FUNCTION_BLOCK CU00xAutomatParalell_1_Task EXTENDS TcoTaskedSequencer 

VAR
	_customTimer: TON;
END_VAR

Run();

(*~
	<docu>
		<summary>
			Main method of the sequener. Custom code needs to be placed here. The sequencer is executed by call of **Instance.Run()** method.
			This method is abstract, and it must be overridden in derived block.
		</summary>
	</docu>
~*)
METHOD PROTECTED Main : BOOL
// Takes mode (step/continous) from the parent controller
THIS^.ModeController.Mode := ParentSequence.ModeController.Mode;

IF (Step(1000, TRUE, 'PARALELL STEP - EXAMPLE OF TIMERS')) THEN
    //-------------------------------------    
		StepCompleteWhen(CurrentStep.Duration >= T#300mS);	
    //-------------------------------------
END_IF
IF (Step(1100, TRUE, 'PARALELL STEP - EXAMPLE OF TIMERS')) THEN
    //-------------------------------------    
		StepCompleteWhen(inCondition:=Timer_1(TRUE,T#100MS));	
    //-------------------------------------
END_IF
IF (Step(1200, TRUE, 'PARALELL STEP - EXAMPLE OF TIMERS')) THEN
    //-------------------------------------    
		StepCompleteWhen(inCondition:=Timer_1(TRUE,T#200MS));	
    //-------------------------------------
END_IF

IF THIS^.IsFreshState THEN
	_customTimer(IN:=FALSE);
END_IF
IF (Step(1300, TRUE, 'PARALELL STEP - EXAMPLE OF TIMERS')) THEN
    //-------------------------------------    

		_customTimer(IN:=TRUE,PT:=T#200MS);
		StepCompleteWhen(inCondition:=_customTimer.Q);	
    //-------------------------------------
END_IF


IF (Step(10000, TRUE, 'PARALELL TASK DONE')) THEN
    //-------------------------------------
    _task.DoneWhen(TRUE );
    //-------------------------------------	
END_IF
END_METHOD

PROPERTY ParentSequence : REFERENCE TO CU00xAutomatTask
GET
VAR
    _parentSequence : POINTER TO CU00xAutomatTask;
END_VAR
IF __QUERYPOINTER(Parent, _parentSequence) THEN 
    ParentSequence REF= _parentSequence^;              
END_IF
END_GET
END_PROPERTY

END_FUNCTION_BLOCK

(* stored: Version 1.1.0.1
   POU CU00xAutomatParalell_1_Task: Id {9100e615-15b9-0e46-102a-be6dd0540361}, SpecialFunc None
   Method Main: Id {738e56f5-b180-0d7a-3d4b-e023b5347a06}
   Property ParentSequence: Id {7ac2da96-928d-01d5-3f41-19bf6253f5f8}
   Get Get: Id {ede87723-a00e-0288-0152-dfa30b58e0ee} *)
